// TIA Portal V20 export
ORGANIZATION_BLOCK "DiagnosticErrorInterrupt"   // OB82, FBD, DiagnosticErrorInterrupt
{ S7_Optimized_Access := 'TRUE' }
// stored: SetENOAutomatically false
   VAR_INPUT
      IO_State : Word;   // IO state of the HW object
      LADDR : HW_ANY;   // Hardware identifier
      Channel : UInt;   // Channel number
      MultiError : Bool;   // =true if more than one error is present
   END_VAR
BEGIN

REGION Network 1: ET200SP 2AQ HF
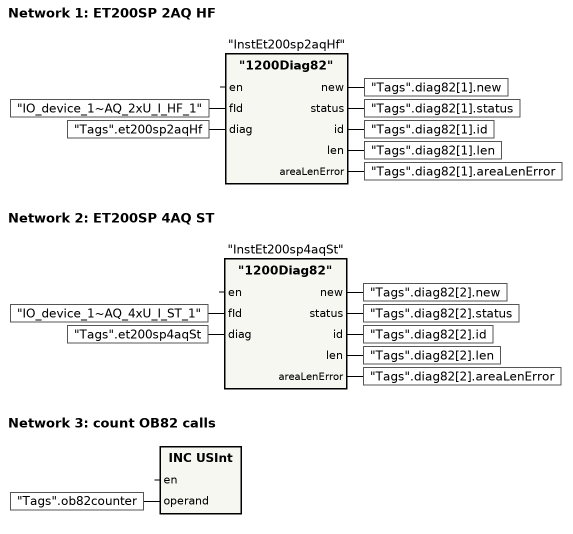
   "InstEt200sp2aqHf"(fId := "IO_device_1~AQ_2xU_I_HF_1",   // "1200Diag82"
                      diag := "Tags".et200sp2aqHf,
                      new => "Tags".diag82[1].new,
                      status => "Tags".diag82[1].status,
                      id => "Tags".diag82[1].id,
                      len => "Tags".diag82[1].len,
                      areaLenError => "Tags".diag82[1].areaLenError);
END_REGION

REGION Network 2: ET200SP 4AQ ST
   "InstEt200sp4aqSt"(fId := "IO_device_1~AQ_4xU_I_ST_1",   // "1200Diag82"
                      diag := "Tags".et200sp4aqSt,
                      new => "Tags".diag82[2].new,
                      status => "Tags".diag82[2].status,
                      id => "Tags".diag82[2].id,
                      len => "Tags".diag82[2].len,
                      areaLenError => "Tags".diag82[2].areaLenError);
END_REGION

REGION Network 3: count OB82 calls
   "Tags".ob82counter := "Tags".ob82counter + 1;
END_REGION
END_ORGANIZATION_BLOCK
